PROGRAM Main_Step_1
VAR
	Always_ON: BOOL;
	Press_Start_Sensor: BOOL;
	Axis04_Press_OFF: TON;
	Test02: BOOL;
	GVL_Main_Step_0: BOOL;
	TEst11: BOOL;
	test111: BOOL;
END_VAR
VAR // added by the converter: edge detectors and wires of the graphical bodies
    _w1, _w2, _w3, _w4, _w5, _w6, _w7, _w8, _w9, _w10, _w11, _w12, _w13 : BOOL;
END_VAR

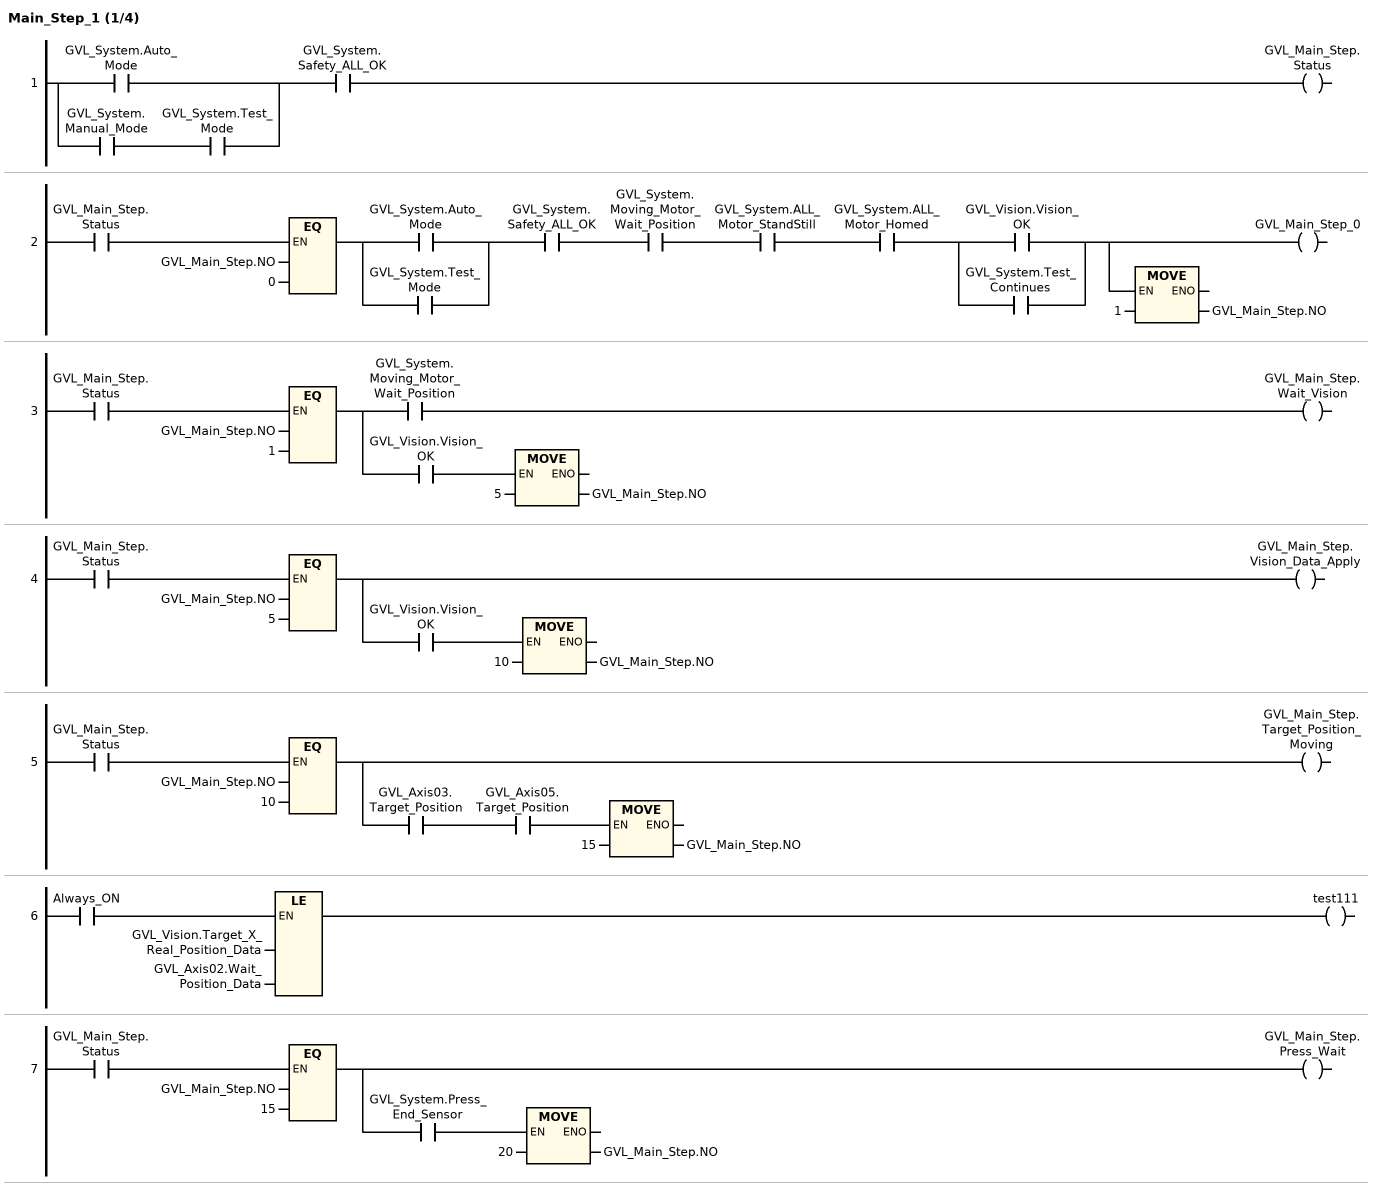
// NETWORK 1
GVL_Main_Step.Status := (GVL_System.Auto_Mode OR GVL_System.Manual_Mode AND GVL_System.Test_Mode) AND GVL_System.Safety_ALL_OK;

// NETWORK 2
_w1 := (GVL_Main_Step.Status AND GVL_Main_Step.NO = 0) AND (GVL_System.Auto_Mode OR GVL_System.Test_Mode) AND GVL_System.Safety_ALL_OK AND GVL_System.Moving_Motor_Wait_Position AND GVL_System.ALL_Motor_StandStill AND GVL_System.ALL_Motor_Homed AND (GVL_Vision.Vision_OK OR GVL_System.Test_Continues);
GVL_Main_Step_0 := _w1;
IF _w1 THEN GVL_Main_Step.NO := 1; END_IF

// NETWORK 3
_w2 := GVL_Main_Step.Status AND GVL_Main_Step.NO = 1;
GVL_Main_Step.Wait_Vision := _w2 AND GVL_System.Moving_Motor_Wait_Position;
IF _w2 AND GVL_Vision.Vision_OK THEN GVL_Main_Step.NO := 5; END_IF

// NETWORK 4
_w3 := GVL_Main_Step.Status AND GVL_Main_Step.NO = 5;
GVL_Main_Step.Vision_Data_Apply := _w3;
IF _w3 AND GVL_Vision.Vision_OK THEN GVL_Main_Step.NO := 10; END_IF

// NETWORK 5
_w4 := GVL_Main_Step.Status AND GVL_Main_Step.NO = 10;
GVL_Main_Step.Target_Position_Moving := _w4;
IF _w4 AND GVL_Axis03.Target_Position AND GVL_Axis05.Target_Position THEN GVL_Main_Step.NO := 15; END_IF

// NETWORK 6
test111 := Always_ON AND GVL_Vision.Target_X_Real_Position_Data <= GVL_Axis02.Wait_Position_Data;

// NETWORK 7
_w5 := GVL_Main_Step.Status AND GVL_Main_Step.NO = 15;
GVL_Main_Step.Press_Wait := _w5;
IF _w5 AND GVL_System.Press_End_Sensor THEN GVL_Main_Step.NO := 20; END_IF

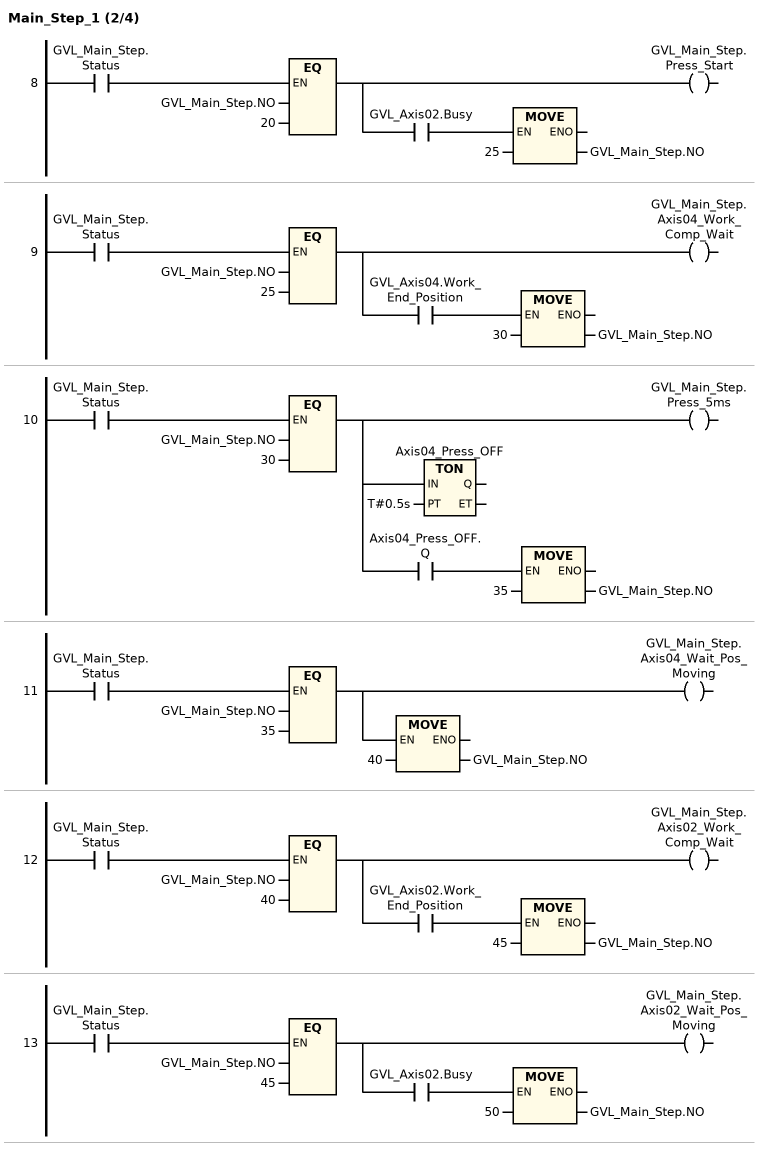
// NETWORK 8
_w6 := GVL_Main_Step.Status AND GVL_Main_Step.NO = 20;
GVL_Main_Step.Press_Start := _w6;
IF _w6 AND GVL_Axis02.Busy THEN GVL_Main_Step.NO := 25; END_IF

// NETWORK 9
_w7 := GVL_Main_Step.Status AND GVL_Main_Step.NO = 25;
GVL_Main_Step.Axis04_Work_Comp_Wait := _w7;
IF _w7 AND GVL_Axis04.Work_End_Position THEN GVL_Main_Step.NO := 30; END_IF

// NETWORK 10
_w8 := GVL_Main_Step.Status AND GVL_Main_Step.NO = 30;
GVL_Main_Step.Press_5ms := _w8;
Axis04_Press_OFF(IN := _w8, PT := T#0.5s); // TON
IF _w8 AND Axis04_Press_OFF.Q THEN GVL_Main_Step.NO := 35; END_IF

// NETWORK 11
_w9 := GVL_Main_Step.Status AND GVL_Main_Step.NO = 35;
GVL_Main_Step.Axis04_Wait_Pos_Moving := _w9;
IF _w9 THEN GVL_Main_Step.NO := 40; END_IF

// NETWORK 12
_w10 := GVL_Main_Step.Status AND GVL_Main_Step.NO = 40;
GVL_Main_Step.Axis02_Work_Comp_Wait := _w10;
IF _w10 AND GVL_Axis02.Work_End_Position THEN GVL_Main_Step.NO := 45; END_IF

// NETWORK 13
_w11 := GVL_Main_Step.Status AND GVL_Main_Step.NO = 45;
GVL_Main_Step.Axis02_Wait_Pos_Moving := _w11;
IF _w11 AND GVL_Axis02.Busy THEN GVL_Main_Step.NO := 50; END_IF

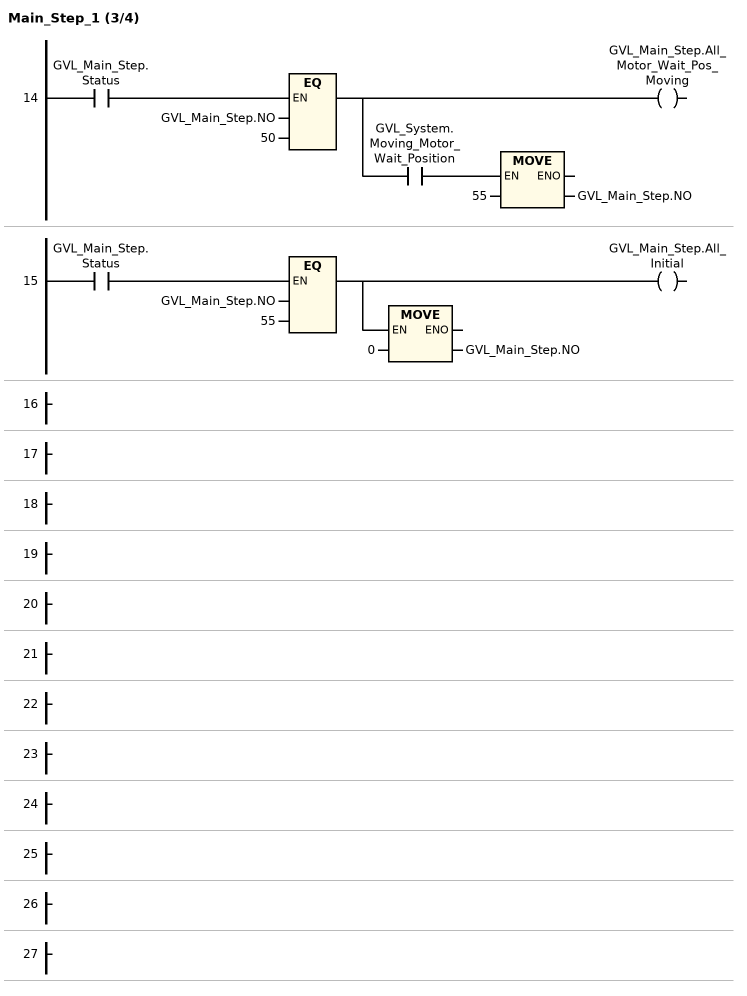
// NETWORK 14
_w12 := GVL_Main_Step.Status AND GVL_Main_Step.NO = 50;
GVL_Main_Step.All_Motor_Wait_Pos_Moving := _w12;
IF _w12 AND GVL_System.Moving_Motor_Wait_Position THEN GVL_Main_Step.NO := 55; END_IF

// NETWORK 15
_w13 := GVL_Main_Step.Status AND GVL_Main_Step.NO = 55;
GVL_Main_Step.All_Initial := _w13;
IF _w13 THEN GVL_Main_Step.NO := 0; END_IF

// NETWORK 16

// NETWORK 17

// NETWORK 18

// NETWORK 19

// NETWORK 20

// NETWORK 21

// NETWORK 22

// NETWORK 23

// NETWORK 24

// NETWORK 25

// NETWORK 26

// NETWORK 27

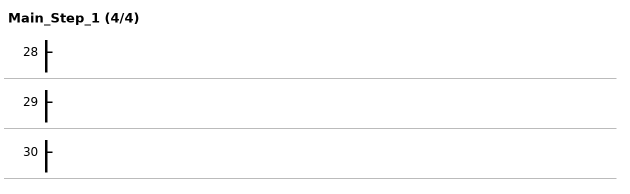
// NETWORK 28

// NETWORK 29

// NETWORK 30

END_PROGRAM

(* stored: Version 1.1.0.1, ProductVersion 3.1.4024.15
   POU Main_Step_1: Id {e9c2e356-0290-4498-93b7-5d71dbb9af9b}, SpecialFunc None *)
